// TIA Portal project "fftia" (V14)

(* hardware
DEVICE "S7-1200 station_1"  S7-1200 Station
   slot 0: "Rack_0"  Rack  V1.0
   slot 1: "PLC_1"  CPU 1214C DC/DC/DC  6ES7 214-1AG40-0XB0  V4.2
*)

// ===== PLC "PLC_1"  CPU 1214C DC/DC/DC =====

VAR_GLOBAL   // PLC tag table "Default tag table"
   "realout" AT %MD100 : Real;
   "ID34_in" AT %MD34 : DWord;
   "xStart" AT %I0.0 : Bool;
   "xMemoryBit_S" AT %M0.0 : Bool;
   "xStop" AT %I0.2 : Bool;
   "X e Stop bit" AT %M0.2 : Bool;
   "xMotor" AT %Q0.0 : Bool;
END_VAR

DATA_BLOCK "mm"   // DB1
{ S7_Optimized_Access := 'TRUE' }
VERSION : 0.1
   VAR
      fft_heartbeat0 : Int;
      fft_heartbeat1 : Int;
      fft_ret_val : Bool;
      indata : Array[0..511] of Real;
      fftmagn : Array[0..511] of Real;
      n_fftsize : Int := 512;
      fftGO : Bool;
      itrend : Int;
      indata_trend : Real;
      fftmagn_trend : Real;
      FFTruntime : Time;
      load_indata : Bool;
      load_1shot : Bool;
      iload : Int;
   END_VAR
BEGIN
   indata[1] := 0.7;
   indata[2] := 1.0;
   indata[3] := 0.7;
   indata[4] := 0.0;
   indata[5] := -0.7;
   indata[6] := -1.0;
   indata[7] := -0.7;
   indata[8] := 0.0;
   indata[9] := 0.7;
   indata[10] := 1.0;
   indata[11] := 0.7;
   indata[12] := 0.0;
   indata[13] := -0.7;
   indata[14] := -1.0;
   indata[15] := -0.7;
   indata[16] := 0.0;
   indata[17] := 0.0;
   indata[18] := 0.0;
   indata[19] := 0.0;
   indata[20] := 0.0;
   indata[21] := 0.0;
   indata[22] := 0.0;
   indata[23] := 0.0;
END_DATA_BLOCK

// folder: System blocks/Program resources

DATA_BLOCK "ffttmr"   // DB2
{ S7_Optimized_Access := 'TRUE' }
AUTHOR : Simatic
FAMILY : IEC
NAME : IEC_TMR
VERSION : 1.0
// stored: InstanceOfName IEC_TIMER
"IEC_TIMER"
BEGIN
END_DATA_BLOCK

// folder: (top level)

FUNCTION "FFT" : Bool   // FC1, SCL
{ S7_Optimized_Access := 'TRUE' }
VERSION : 0.1
   VAR_INPUT
      indata : Array[0..511] of Real;
      n : Int;
   END_VAR
   VAR_OUTPUT
      fftmagn : Array[0..511] of Real;
   END_VAR
   VAR_TEMP
      Areal : Array[0..511] of Real;
      Aimag : Array[0..511] of Real;
      Wreal : Real;
      Wimag : Real;
      WMreal : Real;
      WMimag : Real;
      Treal : Real;
      Timag : Real;
      Ureal : Real;
      "m" : Int;
      halfm : Int;
      kstep : Int;
      jincr : Int;
      kj : Int;
      kjhm : Int;
      ibrs : Array[0..511] of Int;
      itrg : Int;
      isrc : Int;
      iadd : Int;
      ilim : Int;
   END_VAR
   VAR CONSTANT
      U1 : UInt := 1;
   END_VAR
BEGIN
   (* Check Inputs *)
   "mm".fft_heartbeat0 := ("mm".fft_heartbeat0 + 1) AND 4095;
   #FFT := FALSE;
   IF NOT ENO THEN RETURN; END_IF;
   IF #n < 2 THEN RETURN; END_IF;
   IF #n > 512 THEN RETURN; END_IF;
   IF (#n & (#n - 1)) <> 0 THEN RETURN; END_IF;
   "mm".fft_heartbeat1 := ("mm".fft_heartbeat1 + 1) AND 4095;

   (* Start Cooley-Tukey:  bit-reversal; divide and conquer *)

   (* bit-reverse-copy(a, A); indices stored in array ibrs[0..511]     *)
   #ibrs[0] := 0;  (* Seed first index; reversal of index 0 is 0       *)
   #iadd := #n;    (* Seed difference to add                           *)
   #itrg := 1;      (* Start at ibrs[1]                                *)
   WHILE #iadd > 1 DO        (* Loop until next halved iadd would be 0 *)
     #iadd := #iadd / 2;     (* halve iadd i.e. =>256=>...=>1          *)
     #ilim := #n / #iadd;    (* double limit =>2=>4=>...=>512          *)
     #isrc := 0;             (* Start source index at ibrs[0]          *)
     WHILE #itrg < #ilim DO                (* Loop from itrg to ilim-1 *)
       #ibrs[#itrg] := #ibrs[#isrc] + #iadd;  (* Save target index     *)
       #Areal[#itrg] := #indata[#ibrs[#itrg]];(* Copy real data        *)
       #Aimag[#itrg] := 0.0;                  (* Zero out imag data    *)
       #isrc := #isrc + 1;                    (* Next source index     *)
       #itrg := #itrg + 1;                    (* Next target index     *)
     END_WHILE;
   END_WHILE;

   (* Divide and conquer *)

   (* wM <= exp(-2PIi/m) : part 1 of 2; initialization when m is 2 *)
   #WMreal := -1.0; (*  cos(-2PI/m) =  cos(-2PI/2) =  cos(-PI) = -1.0 *)
   #WMimag := 0.0;  (* isin(-2PI/m) = isin(-2PI/2) = isin(-PI) =  0.0 *)

   (* for s = 1 to log(n) : base-2 logarithm *)
   #halfm := 1;
   WHILE #halfm < #n DO
     (* m <= 2^s *)
     #"m" := #halfm * 2;
     (* for k = 0 to n-1 by m : part 1 of 2 *)
     #kstep := 0;
     WHILE #kstep < #n DO
       (* w <= 1 *)
       #Wreal := 1.0;
       #Wimag := 0.0;
       (* for j = 0 to m/2-1 *)
       FOR #jincr := 0 TO (#halfm-1) DO 
         #kj := #kstep + #jincr;
         #kjhm := #kj + #halfm;
         (* t <= w * A[k+j+m/2] *)
         (* u <= A[k+j] : not needed because A[k+j] is last *)
         #Treal := (#Wreal * #Areal[#kjhm]) - (#Wimag * #Aimag[#kjhm]);
         #Timag := (#Wreal * #Aimag[#kjhm]) + (#Wimag * #Areal[#kjhm]);
         (* A[k+j+m/2] <= u - t : use A....[kj] instead of u *)
         #Areal[#kjhm] := #Areal[#kj] - #Treal;
         #Aimag[#kjhm] := #Aimag[#kj] - #Timag;
         (* A[k+j] <= u + t *)
         #Areal[#kj] := #Areal[#kj] + #Treal;
         #Aimag[#kj] := #Aimag[#kj] + #Timag;
         (* w <= w * wM : Ureal holds the new value of Wreal until the *)
         (*               calculation of Wimag using Wreal is complete *)
         #Ureal := (#Wreal * #WMreal) - (#Wimag * #WMimag);
         #Wimag := (#Wreal * #WMimag) + (#Wimag * #WMreal);
         #Wreal := #Ureal;
       END_FOR;
       (* for k = 0 to n=1 by m : part 2 of 2 *)
       #kstep := #kstep + #"m";
     END_WHILE;
     (* Prepare for next pass through the outer while loop             *)
     (* (i) double halfm (m/2), which will double m on next pass start *)
     #halfm := #"m";
     (* (ii) wM <= exp(-2PIi/m) : part 2 of 2, with doubled m          *)
     #WMimag := SQRT((1.0 - #WMreal) / 2.0);
     #WMreal := SQRT((1.0 + #WMreal) / 2.0);
   END_WHILE;                                   (* End of Cooley-Tukey *)

   (* Convert complex DFT to magnitudes N.B. not part of Cooley-Tukey  *)
   FOR #kj := 0 TO (#n-1) DO
       #fftmagn[#kj] := SQRT((#Areal[#kj] * #Areal[#kj]) + (#Aimag[#kj] * #Aimag[#kj]));
   END_FOR;

   #FFT := TRUE;    (* Success *)
END_FUNCTION

FUNCTION "load_indata" : Void   // FC2, SCL
{ S7_Optimized_Access := 'TRUE' }
VERSION : 0.1
   VAR CONSTANT
      twopi : Real := 6.283185;
   END_VAR
BEGIN
   IF "mm".iload > 511 THEN RETURN; END_IF;
   IF "mm".iload >= 0 THEN
       "mm".indata["mm".iload] := (10.0 * SIN("mm".iload * #twopi / (512.0 /  8.00)))
                                + ( 5.0 * COS("mm".iload * #twopi / (512.0 / 17.07)));
   END_IF;
   "mm".iload := "mm".iload + 1;
END_FUNCTION

ORGANIZATION_BLOCK "Main"   // OB1, LAD, ProgramCycle
TITLE = "Main Program"
{ S7_Optimized_Access := 'TRUE' }
VERSION : 0.1
   VAR_INPUT
      Initial_Call : Bool;   // Initial call of this OB
      Remanence : Bool;   // =True, if remanent data are available
   END_VAR
   VAR_TEMP   // added for the SCL form of the ladder/FBD networks
      _w1 : Bool;
      _w2 : Bool;
   END_VAR
BEGIN

REGION Network 1
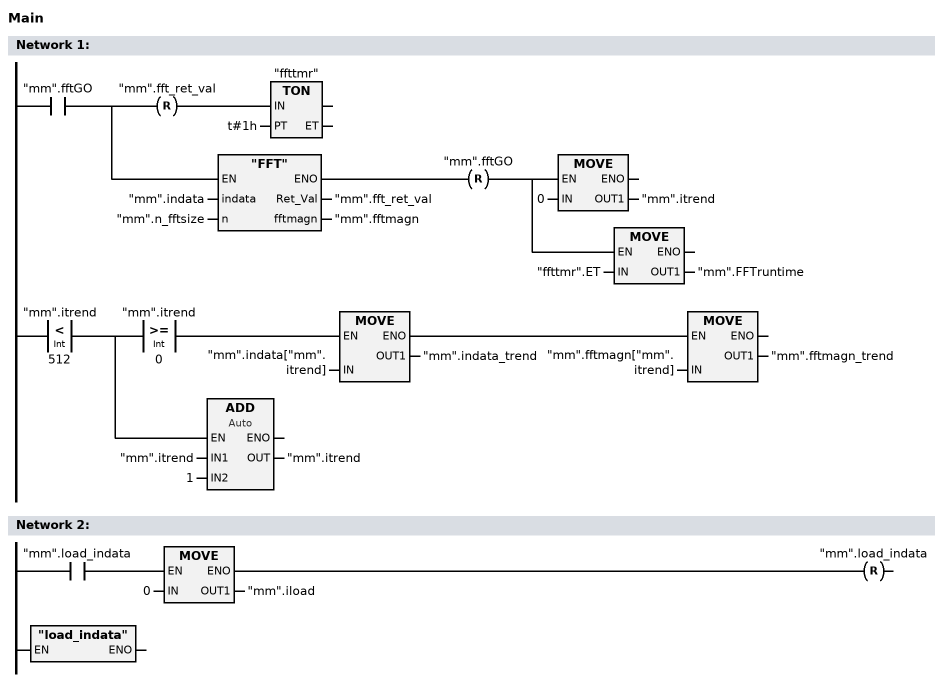
   // ENO of a box is taken as its EN; it also drops when the box reports an error
   IF "mm".fftGO THEN "mm".fft_ret_val := FALSE; END_IF;
   "ffttmr".TON(IN := "mm".fftGO, PT := t#1h);
   "mm".fft_ret_val := "FFT"(EN := "mm".fftGO,
                           indata := "mm".indata,
                           n := "mm".n_fftsize,
                           fftmagn => "mm".fftmagn,
                           ENO => #_w1);
   IF #_w1 THEN
       "mm".fftGO := FALSE;
       "mm".itrend := 0;
       "mm".FFTruntime := "ffttmr".ET;
   END_IF;
   #_w2 := "mm".itrend < 512;
   IF #_w2 AND ("mm".itrend >= 0) THEN
       "mm".indata_trend := "mm".indata["mm".itrend];
       "mm".fftmagn_trend := "mm".fftmagn["mm".itrend];
   END_IF;
   IF #_w2 THEN "mm".itrend := "mm".itrend + 1; END_IF;
END_REGION

REGION Network 2
   RUNG wire#powerrail
      Contact( "mm".load_indata )
      { S7_GenerateENO := "TRUE" } Move(in := 0, out1 => "mm".iload)
      R_Coil( "mm".load_indata )
   END_RUNG
   RUNG wire#powerrail
      "load_indata"()
   END_RUNG
   // the same network as SCL:
   // ENO of a box is taken as its EN; it also drops when the box reports an error
   IF "mm".load_indata THEN
       "mm".iload := 0;
       "mm".load_indata := FALSE;
   END_IF;
   "load_indata"();
END_REGION
END_ORGANIZATION_BLOCK